(* CODESYS project Prova_Ladder.project

Project tree, tasks and I/O mapping:
  Device : CODESYS Control Win V3, 3S - Smart Software Solutions GmbH, order no. 305021, version 3.5.10.30
    application Application
      libraries: Standard, * (System)
      task MainTask (cyclic, interval t#20ms, priority 1) calls PLC_PRG
      task VISU_TASK (cyclic, interval 100 ms, priority 31) calls VisuElems.Visu_Prg
      program PLC_PRG [LD]
      visualisation Visualization
  text list GlobalTextList
*)

// Device/Application/PLC_PRG
PROGRAM PLC_PRG
VAR
	Contact1: BOOL;
	Coil1: BOOL;
END_VAR

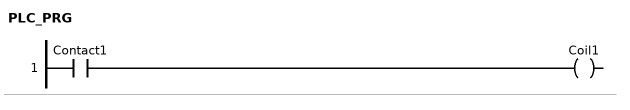
// NETWORK 1
Coil1 := Contact1;

END_PROGRAM

// Device/Application/Visualization
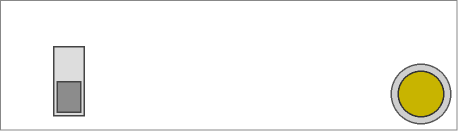
VISUALIZATION Visualization  // 458x131
    DipSwitch (34,46 70x70), variable: PLC_PRG.Contact1, behaviour: TOGGLE, style: Switch-DipSwitch-Gray
    Lamp1 (386,59 70x70), variable: PLC_PRG.Coil1, style: Lamp-Lamp1-Yellow
END_VISUALIZATION
